// TwinCAT 3 PLC project FlyingSaw
// ProgramVersion: 3.1.4023.0
// libraries:
//   Struckig, * (Stefan Besler)
//   Tc3_Module, * (Beckhoff Automation GmbH)
//   ZApplication, 1.5.37.1 (Zeugwerk GmbH)
//   ZEquipment, 1.5.37.1 (Zeugwerk GmbH)
//   ZAux, 1.5.37.1 (Zeugwerk GmbH)
//   ZPlatform, 1.5.37.1 (Zeugwerk GmbH)
//   ZCore, 1.5.37.1 (Zeugwerk GmbH)
// project tree:
//   ZApp/App/ ZApp.TcPOU
//   ZApp/App/_DataTypes/ ZAppStep.TcDUT
//   ZApp/App/_States/ ZAppSequenceBoot.TcPOU, ZAppSequenceBootFault.TcPOU, ZAppSequenceRunning.TcPOU
//   ZApp/App/_SubObjects/ ZAppSequence.TcPOU
//   ZApp/Com/_DataTypes/ BoxesCom.TcDUT, ZCom.TcDUT, ZComUnit.TcDUT
//   ZApp/Data/_DataTypes/ ZData.TcDUT, ZDataMachine.TcDUT, ZDataConfig.TcDUT, ZDataCalibration.TcDUT, ZDataRecipe.TcDUT
//   ZApp/Unit/Machine/ IMachine.TcIO, MachineUnit.TcPOU, MachineUnitProgram.TcPOU
//   ZApp/Unit/Machine/_Com/ MachineCom.TcDUT, MachineComPublish.TcDUT, MachineComPublishEquipment.TcDUT, MachineComRef.TcDUT, MachineComRequest.TcDUT, MachineComSubscribe.TcDUT, MachineComSubscribeEquipment.TcDUT
//   ZApp/Unit/Machine/_DataTypes/ Box.TcDUT, MachineState.TcDUT, MachineStep.TcDUT
//   ZApp/Unit/Machine/_Data/ MachineDataCalibration.TcDUT, MachineDataConfig.TcDUT, MachineDataMachine.TcDUT, MachineDataRef.TcDUT
//   ZApp/Unit/Machine/_Equipment/ MachineActuator.TcPOU, MachineAxis.TcPOU, MachineEquipment.TcPOU, MachineFieldbus.TcPOU, MachineIo.TcPOU, MachineLinkedUnit.TcPOU
//   ZApp/Unit/Machine/_States/ MachineSequenceAutomatic.TcPOU, MachineSequenceBoot.TcPOU, MachineSequenceFaultReaction.TcPOU, MachineSequenceGoHome.TcPOU, MachineSequenceStop.TcPOU
//   ZApp/Unit/Machine/_SubObjects/ BoxRingBuffer.TcPOU, MachineContainer.TcPOU, MachineSequence.TcPOU
//   ZApp/ ZGlobal.TcGVL, ZModuleProgram.TcPOU, ZModuleTask.TcTTO
// real-time tasks:
//   TASK ZModuleTask: cycle T#10ms, priority 20, ADS port 350

CONFIGURATION FlyingSaw
    RESOURCE PLC ON TwinCAT3
        TASK ZModuleTask(INTERVAL := T#10ms, PRIORITY := 20);
        PROGRAM ZModuleProgram WITH ZModuleTask : ZModuleProgram;
    END_RESOURCE
END_CONFIGURATION

// ---- ZApp/App/_DataTypes/ZAppStep.TcDUT
{attribute 'qualified_only'}
{attribute 'to_string'}
TYPE ZAppStep :
(
  Undefined := 0
  
  ,BootBegin
  ,BootLoadDefaultData
  ,BootEnd
  ,BootFaultBegin
  ,BootFaultEnd 
  ,RunningBegin
  ,RunningEnd   
);
END_TYPE

// ---- ZApp/Com/_DataTypes/BoxesCom.TcDUT
TYPE BoxesCom :
STRUCT
  IndexOfFirst : DINT;
  IndexOfNext : DINT;
  Buffer : ARRAY [0..20] OF Box;
END_STRUCT
END_TYPE

// ---- ZApp/Com/_DataTypes/ZCom.TcDUT
TYPE ZCom :
STRUCT
  // module context
  App : ZApplication.ApplicationComPublish;
  Alarming : ZApplication.AlarmingCom;
  Messages : ZApplication.MessagingCom;
  
  // unit context
  Unit : ZComUnit;
  
  Boxes : BoxesCom;

END_STRUCT
END_TYPE

// ---- ZApp/Com/_DataTypes/ZComUnit.TcDUT
TYPE ZComUnit :
STRUCT
{region "Machine"}
{IF NOT (defined (Machine_disabled))}
  Machine : MachineCom;
  {attribute 'ZId' := 'ffcc16ae-32b8-4aad-8514-f391c00062a3'}
{END_IF}
{endregion}
{attribute '__ZwPlcApplicationComUnitDeclaration__'} // Do not remove this attribute! It is used for code generation.
END_STRUCT
END_TYPE

// ---- ZApp/Data/_DataTypes/ZData.TcDUT
TYPE ZData :
STRUCT
  Config : ZDataConfig;
  Machine : ZDataMachine;
  Calibration : ZDataCalibration;
  Recipe : ZDataRecipe;
END_STRUCT
END_TYPE

// ---- ZApp/Data/_DataTypes/ZDataMachine.TcDUT
TYPE ZDataMachine :
STRUCT
{region "Machine"}
{IF NOT (defined (Machine_disabled))}
  Machine : MachineDataMachine;
  {attribute 'ZId' := 'ffcc16ae-32b8-4aad-8514-f391c00062a3'}
{END_IF}
{endregion}
{attribute '__ZwPlcApplicationDataMachineDeclaration__'} // Do not remove this attribute! It is used for code generation.
END_STRUCT
END_TYPE

// ---- ZApp/Data/_DataTypes/ZDataConfig.TcDUT
TYPE ZDataConfig :
STRUCT
{region "Machine"}
{IF NOT (defined (Machine_disabled))}
  Machine : MachineDataConfig;
  {attribute 'ZId' := 'ffcc16ae-32b8-4aad-8514-f391c00062a3'}
{END_IF}
{endregion}
{attribute '__ZwPlcApplicationDataConfigDeclaration__'} // Do not remove this attribute! It is used for code generation.
END_STRUCT
END_TYPE

// ---- ZApp/Data/_DataTypes/ZDataCalibration.TcDUT
TYPE ZDataCalibration :
STRUCT
{region "Machine"}
{IF NOT (defined (Machine_disabled))}
  Machine : MachineDataCalibration;
  {attribute 'ZId' := 'ffcc16ae-32b8-4aad-8514-f391c00062a3'}
{END_IF}
{endregion}
{attribute '__ZwPlcApplicationDataCalibrationDeclaration__'} // Do not remove this attribute! It is used for code generation.
END_STRUCT
END_TYPE

// ---- ZApp/Data/_DataTypes/ZDataRecipe.TcDUT
TYPE ZDataRecipe :
STRUCT
  RecipeParam1 : LREAL;
  RecipeParam2 : LREAL;
  RecipeParam3 : LREAL;
END_STRUCT
END_TYPE

// ---- ZApp/Unit/Machine/_Com/MachineCom.TcDUT
/// This struct contains variables that
/// * are read from outside (e.g. HMI) to retrieve information about the unit's current state and (temporary) parameters (= `publish`) 
/// * are written from outside (e.g. HMI) to control the unit via ADS (= `subscribe`) 
TYPE MachineCom :
STRUCT
  Publish : MachineComPublish;
  Subscribe : MachineComSubscribe;
END_STRUCT
END_TYPE

// ---- ZApp/Unit/Machine/_Com/MachineComPublish.TcDUT
/// this is the container of informations that the unit wants to share with the world outside of the PLC
/// This struct should only be read from by external applications.
TYPE MachineComPublish :
STRUCT
  State : ZApplication.UnitStateMachineState; // state the unit is in
  Request : MachineComRequest; // booleans that indictate which action is currently possible to perform with this unit
  Equipment : MachineComPublishEquipment;  // structs for equipment objects which are used by the bridges
END_STRUCT
END_TYPE

// ---- ZApp/Unit/Machine/_Com/MachineComPublishEquipment.TcDUT
TYPE MachineComPublishEquipment :
STRUCT

{region "TransportX : Axis"}
  TransportX : ZApplication.AxisComPublish;
  {attribute 'ZId' := 'e985697b-7ba2-4e1b-acce-25e7c1308b60'}
{endregion}

{region "ToolX : Axis"}
  ToolX : ZApplication.AxisComPublish;
  {attribute 'ZId' := '805b377d-816e-493b-a105-09954c5e25a1'}
{endregion}

{attribute '__ZwPlcUnitComDeclaration__'} // Do not remove this attribute! It is used for code generation.

END_STRUCT
END_TYPE

// ---- ZApp/Unit/Machine/_Com/MachineComRef.TcDUT
/// container for all communication data types that are used by the unit
TYPE MachineComRef :
STRUCT
  Publish : REFERENCE TO MachineComPublish; 
  Subscribe : REFERENCE TO MachineComSubscribe; 
END_STRUCT
END_TYPE

// ---- ZApp/Unit/Machine/_Com/MachineComRequest.TcDUT
TYPE MachineComRequest :
STRUCT
  Start : BOOL;
  Stop : BOOL;
  GoHome : BOOL;
  Halt : BOOL;
END_STRUCT
END_TYPE

// ---- ZApp/Unit/Machine/_Com/MachineComSubscribe.TcDUT
TYPE MachineComSubscribe :
STRUCT
  Request : MachineComRequest; // contains booleans that are used to start a specific sequence.
  Equipment : MachineComSubscribeEquipment;  // structs for equipment objects which are used by the bridges
END_STRUCT
END_TYPE

// ---- ZApp/Unit/Machine/_Com/MachineComSubscribeEquipment.TcDUT
TYPE MachineComSubscribeEquipment :
STRUCT

{region "TransportX : Axis"}
  TransportX : ZApplication.AxisComSubscribe;
  {attribute 'ZId' := 'e985697b-7ba2-4e1b-acce-25e7c1308b60'}
{endregion}

{region "ToolX : Axis"}
  ToolX : ZApplication.AxisComSubscribe;
  {attribute 'ZId' := '805b377d-816e-493b-a105-09954c5e25a1'}
{endregion}

{region "BoxDetected : Digital"}
  BoxDetected : ZApplication.DigitalComSubscribe;
  {attribute 'ZId' := 'd9755a0b-6503-481c-99e0-54f892b6c08c'}
{endregion}

{attribute '__ZwPlcUnitComDeclaration__'} // Do not remove this attribute! It is used for code generation.

END_STRUCT
END_TYPE

// ---- ZApp/Unit/Machine/_DataTypes/Box.TcDUT
TYPE Box :
STRUCT
  BoxId : INT;
  DetectedAt : LWORD;
  CompletionRatio : LREAL;
END_STRUCT
END_TYPE

// ---- ZApp/Unit/Machine/_DataTypes/MachineState.TcDUT
/// This enumeration contains all used defined sequences of a unit.
/// Per default a unit makes use of the states that are contained in (UnitStateDefault)[xref:ZApplication.UnitStateDefault]. However,
/// most of the time a unit need to perform some application depend sequences that can be performed by putting the unit into userdefined states.
/// For instance, a robotic unit could use the state (automatic)[xref:ZApplication.UnitStateDefault] to lift an object from point A to point B,
/// a userdefined state could be used to open and close the robotic-units gripper, respectively
{attribute 'qualified_only'}
TYPE MachineState :
(
	UserdefinedState1 := ZApplication.UnitStateMachineState.Last+1
);
END_TYPE

// ---- ZApp/Unit/Machine/_DataTypes/MachineStep.TcDUT
/// This enumeration contains all steps that are used by the various sequences of a unit.
/// Sequences use a subrange (***Begin to ***End) of this enumeration.
{attribute 'qualified_only'}
{attribute 'to_string'}
TYPE MachineStep :
(
  Undefined := 0
  
  ,BootBegin
  ,BootEnd 

  ,StopBegin
  ,StopEnd

  ,AutomaticBegin
  ,AutomaticRunTool
  ,AutomaticEnd
  
  ,GoHomeBegin
  ,GoHomeEnd 
  
  ,FaultReactionBegin
  ,FaultReactionEnd
);
END_TYPE

// ---- ZApp/Unit/Machine/_Data/MachineDataCalibration.TcDUT
/// calibration that is determined by calibration sequences of the unit (static offsets, shifts)
TYPE MachineDataCalibration :
STRUCT
END_STRUCT
END_TYPE

// ---- ZApp/Unit/Machine/_Data/MachineDataConfig.TcDUT
/// configuration data that is used during boot to configure the Units equipment
TYPE MachineDataConfig :
STRUCT
  Simulated : BOOL;
END_STRUCT
END_TYPE

// ---- ZApp/Unit/Machine/_Data/MachineDataMachine.TcDUT
/// machine data that is used through most sequences of the unit (motor speed, axes positions, ...)
TYPE MachineDataMachine :
STRUCT
  Slowspeed : LREAL;
  Highspeed : LREAL;
END_STRUCT
END_TYPE

// ---- ZApp/Unit/Machine/_Data/MachineDataRef.TcDUT
/// container for all data that are used by the unit
TYPE MachineDataRef :
STRUCT
  Config : REFERENCE TO MachineDataConfig; // data required for booting the unit (axes configuration, simulation, parameters that have to be written in PREOP, ...)
  Machine : REFERENCE TO MachineDataMachine; // speeds, positions, ...
  Calibration : REFERENCE TO MachineDataCalibration; // offsets, shifts of nominal to actual values
END_STRUCT
END_TYPE

// ---- ZApp/ZGlobal.TcGVL
{attribute 'qualified_only'}
VAR_GLOBAL
  Com : ZCom;
END_VAR
VAR_GLOBAL PERSISTENT
  Data : ZData;
END_VAR

// ---- ZApp/Unit/Machine/IMachine.TcIO
INTERFACE IMachine EXTENDS ZApplication.IUnit

END_INTERFACE

// ---- ZApp/ZModuleProgram.TcPOU
/// Zeugwerk Application
PROGRAM ZModuleProgram
VAR_INPUT
{region "ZModuleProgram : Utility"}
  App : ZApp(displayName:='Zeugwerk-Application Template', com:=ZGlobal.Com.App);
  Datetime : ZAux.DateTimeUM;
  {attribute 'ZId' := ''}
{endregion}
{region "ZModuleProgram : Logging"}
  Alarming : ZApplication.Alarming(App, datetime := Datetime, com := ZGlobal.Com.Alarming);
  LoggerHmi : ZApplication.Messaging(App, datetime := Datetime, com := ZGlobal.Com.Messages);
  LoggerFile : ZAux.LoggerFile7FF(App, datetime := Datetime, filePath:='C:\Zeugwerk\logs\messages.log', target:='');
  Logger : ZAux.Logging;
  {attribute 'ZId' := ''}
{endregion}  
{attribute '__ZwPlcApplicationModuleProgramDeclaration__'} // Do not remove this attribute! It is used for code generation.
{region "Machine"}
{undefine RunInSeparateProgram}
{IF NOT (defined (Machine_disabled)) AND NOT (defined (RunInSeparateProgram))}
  Machine : MachineUnit(name := 'Machine', // name of the unit (for logging)
					  parent := App, // caller of the Unit's cyclic method. If the Unit runs in its own context use 0
						configdata := ZGlobal.Data.Config.Machine,
						machinedata := ZGlobal.Data.Machine.Machine,
						calibrationdata := ZGlobal.Data.Calibration.Machine,
						com := ZGlobal.Com.Unit.Machine);
  {attribute 'section' := '__ZwPlcUnitProgramDeclaration__'}
  {attribute 'ZId' := 'ffcc16ae-32b8-4aad-8514-f391c00062a3'}
{END_IF}
{endregion}
{attribute '__ZwPlcUnitProgramDeclaration__'} // Do not remove this attribute! It is used for code generation.
END_VAR

{region "ZModuleProgram : Utility"}
  Datetime.Cyclic();
  App.Cyclic();
  {attribute 'ZId' := ''}
{endregion}
{attribute '__ZwPlcApplicationModuleProgramImplementation__'} // Do not remove this attribute! It is used for code generation.

END_PROGRAM

// ---- ZApp/App/ZApp.TcPOU
FUNCTION_BLOCK ZApp EXTENDS ZApplication.Application
VAR
  _boot : ZAppSequenceBoot;
  _bootFault : ZAppSequenceBootFault;
  _running : ZAppSequenceRunning;
END_VAR

METHOD FB_init : BOOL
VAR_INPUT
  bInitRetains : BOOL; /// if TRUE, the retain variables are initialized (warm start / cold start)
  bInCopyCode : BOOL; /// if TRUE, the instance afterwards gets moved into the copy code (online change)
  displayName : ZCore.ZString;
  com : REFERENCE TO ZApplication.ApplicationComPublish;
END_VAR
SetBootSequence(_boot);
SetBootFaultSequence(_bootFault);
SetRunningSequence(_running);
END_METHOD

END_FUNCTION_BLOCK

// ---- ZApp/App/_States/ZAppSequenceBoot.TcPOU
FUNCTION_BLOCK ZAppSequenceBoot EXTENDS ZAppSequence IMPLEMENTS ZCore.ISequence
VAR
  _step : ZCore.Step(ZAppStep.BootBegin, ZAppStep.BootEnd);
END_VAR

IF OnStart(_step)
THEN
  // init custom sequence variables here ...
END_IF

REPEAT
  LogStep();

  CASE _step.Index OF
    (* -------------------------------------------------------------------------------------------------------------------------------- *)
    ZAppStep.BootBegin:
    (* -------------------------------------------------------------------------------------------------------------------------------- *)
    
      IF _step.OnEntry()
      THEN
        ZModuleProgram.LoggerFile.MinimumLevel := ZCore.LogLevel.Trace;
        ZModuleProgram.Logger.AddLogger(ZModuleProgram.LoggerFile);        
        {attribute '__ZwPlcAppZComModuleContext__'} // Do not remove this attribute! It is used for code generation.      
      END_IF
      
	  IF ZModuleProgram.Datetime.State <> ZCore.ObjectState.Booting
      THEN
        _step.SetNext(ZAppStep.BootLoadDefaultData);        
      END_IF
      
    (* -------------------------------------------------------------------------------------------------------------------------------- *)
    ZAppStep.BootLoadDefaultData:
    (* -------------------------------------------------------------------------------------------------------------------------------- *)

      {warning 'The application is loading the default config data on every restart!'}
      LoadDefaultConfigData();
      
      IF IsCommissioning()
      THEN
        LoadDefaultData();
      END_IF
      
      _step.SetNext(ZAppStep.BootEnd);
      
    (* -------------------------------------------------------------------------------------------------------------------------------- *)
    ZAppStep.BootEnd:
    (* -------------------------------------------------------------------------------------------------------------------------------- *)
      SetBusy(FALSE);
      
  ELSE
    Abort('sequence contains unhandled step');
  END_CASE
UNTIL _step.IsNotRepeatable() OR_ELSE NOT Busy END_REPEAT

METHOD  IsCommissioning : BOOL
IsCommissioning := TRUE;
END_METHOD

METHOD FINAL LoadDefaultConfigData

{region "Machine"}
  {IF NOT (defined (Machine_disabled))}
  ZGlobal.Data.Config.Machine.Simulated := TRUE;
  {region "UserInitCode"}
  // put your individual init code for this unit here
  {endregion}
  {END_IF}
  {attribute 'ZId' := 'ffcc16ae-32b8-4aad-8514-f391c00062a3'}
{endregion}

{attribute '__ZwPlcUnitLoadDefaultConfigData__'} // Do not remove this attribute! It is used for code generation.
END_METHOD

METHOD FINAL LoadDefaultData

{attribute '__ZwPlcUnitLoadDefaultData__'} // Do not remove this attribute! It is used for code generation.
END_METHOD

END_FUNCTION_BLOCK

// ---- ZApp/App/_SubObjects/ZAppSequence.TcPOU
FUNCTION_BLOCK ABSTRACT ZAppSequence EXTENDS ZApplication.Sequence IMPLEMENTS ZCore.ISequence

METHOD StepDecoded : ZCore.ZString
VAR_INPUT
  stepIndex : INT;
END_VAR
VAR_INST
  _stepIndexDecoded : ZAppStep;
END_VAR
_stepIndexDecoded := stepIndex;
StepDecoded := TO_STRING(_stepIndexDecoded);
END_METHOD

END_FUNCTION_BLOCK

// ---- ZApp/App/_States/ZAppSequenceBootFault.TcPOU
FUNCTION_BLOCK ZAppSequenceBootFault EXTENDS ZAppSequence IMPLEMENTS ZCore.ISequence
VAR
  _step : ZCore.Step(ZAppStep.BootFaultBegin, ZAppStep.BootFaultEnd);
END_VAR

IF OnStart(_step)
THEN
  // init custom sequence variables here ...
END_IF

REPEAT
  LogStep();

  CASE _step.Index OF
    (* -------------------------------------------------------------------------------------------------------------------------------- *)
    ZAppStep.BootFaultBegin:
    (* -------------------------------------------------------------------------------------------------------------------------------- *)
      _step.SetNext(ZAppStep.BootFaultEnd);
      
    (* -------------------------------------------------------------------------------------------------------------------------------- *)
    ZAppStep.BootFaultEnd:
    (* -------------------------------------------------------------------------------------------------------------------------------- *)
      SetBusy(FALSE);
      
  ELSE
    Abort('sequence contains unhandled step');
  END_CASE
UNTIL _step.IsNotRepeatable() OR_ELSE NOT Busy END_REPEAT

END_FUNCTION_BLOCK

// ---- ZApp/App/_States/ZAppSequenceRunning.TcPOU
FUNCTION_BLOCK ZAppSequenceRunning EXTENDS ZAppSequence IMPLEMENTS ZCore.ISequence
VAR
  _step : ZCore.Step(ZAppStep.RunningBegin, ZAppStep.RunningEnd);
END_VAR

IF OnStart(_step)
THEN
  // init custom sequence variables here ...
END_IF

REPEAT
  LogStep();

  CASE _step.Index OF
    (* -------------------------------------------------------------------------------------------------------------------------------- *)
    ZAppStep.RunningBegin:
    (* -------------------------------------------------------------------------------------------------------------------------------- *)
      ; // implement me
      
    (* -------------------------------------------------------------------------------------------------------------------------------- *)
    ZAppStep.RunningEnd:
    (* -------------------------------------------------------------------------------------------------------------------------------- *)
      SetBusy(FALSE);
      
  ELSE
    Abort('sequence contains unhandled step');
  END_CASE
UNTIL _step.IsNotRepeatable() OR_ELSE NOT Busy END_REPEAT

END_FUNCTION_BLOCK

// ---- ZApp/Unit/Machine/MachineUnit.TcPOU
/// Declaration of a distinct unit of this application
FUNCTION_BLOCK MachineUnit EXTENDS ZApplication.Unit IMPLEMENTS IMachine
VAR
  _equipment : MachineEquipment(THIS^);
  _data : MachineDataRef;
  _com : MachineComRef;

  _boot : MachineSequenceBoot(THIS^);
  _automatic : MachineSequenceAutomatic(THIS^);
  _stop : MachineSequenceStop(THIS^);
  _gohome : MachineSequenceGoHome(THIS^);
  _faultReaction : MachineSequenceFaultReaction(THIS^);
  
  _statemachine : ZApplication.UnitStateMachine;

  _observeTimer : ZAux.Timer; 
END_VAR

{attribute 'ZId' := '7a669cb2-1530-4a61-a6bf-785d936ff64f'}

IF _observeTimer.Done THEN
  _observeTimer.WaitAsync(0.1);
  
  // monitor _com for requested actions (e.g. start homing, start automatic mode, ...)
  ObserveRequest(_com.Subscribe.Request.Start, ZApplication.UnitStateMachineState.Automatic);
  ObserveRequest(_com.Subscribe.Request.Stop, ZApplication.UnitStateMachineState.Stop);
  ObserveRequest(_com.Subscribe.Request.GoHome, ZApplication.UnitStateMachineState.GoHome);
  ObserveRequest(_com.Subscribe.Request.Halt, ZApplication.UnitStateMachineState.Halt);
  
  // provide relevant information via ADS
  _com.Publish.Request.Stop := _stateMachine.IsTransitionAllowed(ZApplication.UnitStateMachineState.Stop);
  _com.Publish.Request.Start := _stateMachine.IsTransitionAllowed(ZApplication.UnitStateMachineState.Automatic);
  _com.Publish.Request.GoHome := _stateMachine.IsTransitionAllowed(ZApplication.UnitStateMachineState.GoHome);
  _com.Publish.Request.Halt := _stateMachine.IsTransitionAllowed(ZApplication.UnitStateMachineState.Halt);

  _com.Publish.State := _stateMachine.State();
END_IF

METHOD FB_init : BOOL
VAR_INPUT
  bInitRetains : BOOL; // if TRUE, the retain variables are initialized (warm start / cold start)
  bInCopyCode : BOOL;  // if TRUE, the instance afterwards gets moved into the copy code (online change)
  parent : ZCore.IManagedObject; // caller of the Unit's cyclic method. If the Unit runs in its own context use 0
  name : ZCore.ZString;  // name of this unit as it should show up in the logger
  configdata : REFERENCE TO MachineDataConfig;  // reference to the configuration data that is used during boot to configure the Units equipment
  machinedata : REFERENCE TO MachineDataMachine; // reference to the machine data that is used through most sequences of the unit (motor speed, axes positions, ...)
  calibrationdata : REFERENCE TO MachineDataCalibration;  // reference to calibration that is determined by calibration sequences of the unit (static offsets, shifts)
  com : REFERENCE TO MachineCom;  // reference to the communication interface that is used to control this Unit via ADS
END_VAR
_name := name;

// initialize local logger decorator
_loggerDecorator.FB_init(bInitRetains, bInCopyCode, name, ZModuleProgram.Logger);
_alarmingDecorator.FB_init(bInitRetains, bInCopyCode, name, ZModuleProgram.Alarming);

// setup data
_data.Config REF= configdata;
_data.Machine REF= machinedata;
_data.Calibration REF= calibrationdata;
_com.Publish REF= com.Publish;
_com.Subscribe REF= com.Subscribe;

// ------- sequence initialization, map sequences of this unit to the statemachine -------
{attribute '__ZwPlcUnitInitSequenceImplementation__'} // Do not remove this attribute! It is used for code generation.
_statemachine.SetSequence(ZApplication.UnitStateMachineState.Boot, _boot);
_statemachine.SetSequence(ZApplication.UnitStateMachineState.FaultReaction, _faultReaction);
_statemachine.SetSequence(ZApplication.UnitStateMachineState.Gohome, _gohome);
_statemachine.SetSequence(ZApplication.UnitStateMachineState.Stop, _stop);
_statemachine.SetSequence(ZApplication.UnitStateMachineState.Automatic, _automatic);

_statemachine.SetName(_name);
_statemachine.SetLogger(_logger);

// set initial state
_statemachine.SetState(ZApplication.UnitStateMachineState.Boot);
SetStateMachine(_statemachine);
END_METHOD

END_FUNCTION_BLOCK

// ---- ZApp/Unit/Machine/_Equipment/MachineEquipment.TcPOU
/// This function block is a container for equipment that is used by this unit.
/// Equipment is grouped by its kind (actuator, axes, io, ...).
/// It extends from [ManagedObjectContainer](xref:ZCore.ManagedObjectContainer) such that the parent
/// (= the unit itself) can be passed to equipment instances.
FUNCTION_BLOCK MachineEquipment EXTENDS MachineContainer
VAR_INPUT
  Io : MachineIo(_parent);
  Actuator : MachineActuator(_parent);
  Axis : MachineAxis(_parent);
  Fieldbus : MachineFieldbus(_parent);
  Unit : MachineLinkedUnit(_parent);
END_VAR

END_FUNCTION_BLOCK

// ---- ZApp/Unit/Machine/_SubObjects/MachineContainer.TcPOU
FUNCTION_BLOCK MachineContainer EXTENDS ZCore.ObjectContainer
VAR_INPUT
END_VAR
VAR_OUTPUT
END_VAR
VAR
  {attribute 'hide'}
  _parent : REFERENCE TO MachineUnit;
END_VAR

{attribute 'hide' }
METHOD FB_init : BOOL
VAR_INPUT
	bInitRetains : BOOL; // if TRUE, the retain variables are initialized (warm start / cold start)
	bInCopyCode : BOOL;  // if TRUE, the instance afterwards gets moved into the copy code (online change)
  unit : REFERENCE TO MachineUnit;
END_VAR
_parent REF= unit;
END_METHOD

END_FUNCTION_BLOCK

// ---- ZApp/Unit/Machine/_Equipment/MachineIo.TcPOU
/// This function block is a container for all I/Os that are used by this unit.
/// The parent of all objects can be directly transfered in their constructor (this is only relevant for equipment objects
/// that have to be managed (e.g. [DebouncedInput](xref:ZEquipment.DebouncedInput), [Light](xref:ZEquipment.Light), ...).
FUNCTION_BLOCK MachineIo EXTENDS MachineContainer
VAR
  {attribute 'hide'}
  _iobridge : ZApplication.IoBridge(_parent);
END_VAR
VAR_INPUT

{region "BoxDetected : DigitalInput"}
  BoxDetected : ZEquipment.DigitalInput;
  {attribute 'ZId' := 'd9755a0b-6503-481c-99e0-54f892b6c08c'}
{endregion}

{attribute '__ZwPlcUnitEquipmentDeclaration__'} // Do not remove this attribute! It is used for code generation.
END_VAR

IF _isInitialized
THEN
  RETURN;
END_IF

  _iobridge.SetLogger(_parent._logger);

{region "BoxDetected : DigitalInput"}
  BoxDetected.SetLogger(_parent._logger);
  BoxDetected.SetName('BoxDetected');
  BoxDetected.SetSimulation(on:=_parent._data.Config.Simulated);
  BoxDetected.SetLogic(ZEquipment.DigitalLogic.Normal);
  _ioBridge.AddDigitalInput(BoxDetected, publish := _parent._com.Publish.Equipment.BoxDetected, subscribe := _parent._com.Subscribe.Equipment.BoxDetected);

  {region "UserInitCode"}
  // put your individual init code for this I/O here
  {endregion}

  {attribute 'ZId' := 'd9755a0b-6503-481c-99e0-54f892b6c08c'}
{endregion}

{attribute '__ZwPlcUnitEquipmentImplementation__'} // Do not remove this attribute! It is used for code generation.

_isInitialized := TRUE;

END_FUNCTION_BLOCK

// ---- ZApp/Unit/Machine/_Equipment/MachineActuator.TcPOU
/// This function block is a container for all actuator objects that are used by this unit.
/// The parent of all objects can be directly transfered in their constructor (this is only relevant for equipment objects
/// that have to be managed (e.g. [DebouncedInput](xref:ZEquipment.DebouncedInput), [Light](xref:ZEquipment.Light), ...).
FUNCTION_BLOCK MachineActuator EXTENDS MachineContainer
VAR
  {attribute 'hide'}
  _actuatorbridge : ZApplication.ActuatorBridge(_parent);
  {attribute 'hide'}
  _iobridge : ZApplication.IoBridge(_parent);
END_VAR
VAR_INPUT

{attribute '__ZwPlcUnitEquipmentDeclaration__'} // Do not remove this attribute! It is used for code generation.
END_VAR

IF _isInitialized
THEN
  RETURN;
END_IF

  _actuatorbridge.SetLogger(_parent._logger);

{attribute '__ZwPlcUnitEquipmentImplementation__'} // Do not remove this attribute! It is used for code generation.

_isInitialized := TRUE;

END_FUNCTION_BLOCK

// ---- ZApp/Unit/Machine/_Equipment/MachineAxis.TcPOU
/// This function block is a container for all axis objects that are used by this unit.
/// The parent of all objects can be directly transfered in their constructor (this is only relevant for equipment objects
/// that have to be managed (e.g. [DebouncedInput](xref:ZEquipment.DebouncedInput), [Light](xref:ZEquipment.Light), ...).
FUNCTION_BLOCK MachineAxis EXTENDS MachineContainer
VAR
  {attribute 'hide'}
  _axisbridge : ZApplication.AxisBridge(_parent);
END_VAR
VAR_INPUT

{region "TransportX : AxisPlcOpenMc"}
  TransportX : ZEquipment.AxisSimulated(_parent);
  {attribute 'ZId' := 'e985697b-7ba2-4e1b-acce-25e7c1308b60'}
{endregion}

{region "ToolX : AxisPlcOpenMc"}
  ToolX : ZEquipment.AxisSimulated(_parent);
  {attribute 'ZId' := '805b377d-816e-493b-a105-09954c5e25a1'}
{endregion}

{attribute '__ZwPlcUnitEquipmentDeclaration__'} // Do not remove this attribute! It is used for code generation.
END_VAR

IF _isInitialized
THEN
  RETURN;
END_IF

  _axisbridge.SetLogger(_parent._logger);

{region "TransportX : AxisPlcOpenMc"}
  TransportX.SetLogger(_parent._logger);
  TransportX.SetName(name:='TransportX');
  TransportX.SetSimulation(_parent._data.Config.Simulated);
  _axisbridge.WithHoming(TransportX)
     .WithMovePosition(TransportX)
     .WithMoveVelocity(TransportX)
     .WithHalt(TransportX)
     .WithVelocityFeedrate(TransportX)
     .WithFeedbackPosition(TransportX)
     .WithFeedbackVelocity(TransportX)
     .WithFeedbackCurrent(TransportX)
     .AddAxis (axis:=TransportX, publish:=_parent._com.Publish.Equipment.TransportX, subscribe:=_parent._com.Subscribe.Equipment.TransportX);


  {region "UserInitCode"}
  // put your individual init code for this Axis here
  {endregion}

  {attribute 'ZId' := 'e985697b-7ba2-4e1b-acce-25e7c1308b60'}
{endregion}

{region "ToolX : AxisPlcOpenMc"}
  ToolX.SetLogger(_parent._logger);
  ToolX.SetName(name:='ToolX');
  ToolX.SetSimulation(_parent._data.Config.Simulated);
  _axisbridge.WithHoming(ToolX)
     .WithMovePosition(ToolX)
     .WithMoveVelocity(ToolX)
     .WithHalt(ToolX)
     .WithVelocityFeedrate(ToolX)
     .WithFeedbackPosition(ToolX)
     .WithFeedbackVelocity(ToolX)
     .WithFeedbackCurrent(ToolX)
     .AddAxis (axis:=ToolX, publish:=_parent._com.Publish.Equipment.ToolX, subscribe:=_parent._com.Subscribe.Equipment.ToolX);

  {region "UserInitCode"}
  // put your individual init code for this Axis here
  {endregion}

  {attribute 'ZId' := '805b377d-816e-493b-a105-09954c5e25a1'}
{endregion}

{attribute '__ZwPlcUnitEquipmentImplementation__'} // Do not remove this attribute! It is used for code generation.

_isInitialized := TRUE;

END_FUNCTION_BLOCK

// ---- ZApp/Unit/Machine/_Equipment/MachineFieldbus.TcPOU
/// This function block is a container for all axis objects that are used by this unit.
/// The parent of all objects can be directly transfered in their constructor (this is only relevant for equipment objects
/// that have to be managed (e.g. [DebouncedInput](xref:ZEquipment.DebouncedInput), [Light](xref:ZEquipment.Light), ...).
FUNCTION_BLOCK MachineFieldbus EXTENDS MachineContainer
VAR
END_VAR
VAR_INPUT

{attribute '__ZwPlcUnitEquipmentDeclaration__'} // Do not remove this attribute! It is used for code generation.
END_VAR

IF _isInitialized
THEN
  RETURN;
END_IF

{attribute '__ZwPlcUnitEquipmentImplementation__'} // Do not remove this attribute! It is used for code generation.

_isInitialized := TRUE;

END_FUNCTION_BLOCK

// ---- ZApp/Unit/Machine/_Equipment/MachineLinkedUnit.TcPOU
/// This function block is a container for all linked units that are used by this unit.
/// Linked units can be addressed through their individual interface.
FUNCTION_BLOCK MachineLinkedUnit EXTENDS MachineContainer
VAR_INPUT
{attribute '__ZwPlcUnitEquipmentDeclaration__'} // Do not remove this attribute! It is used for code generation.
END_VAR

IF _isInitialized
THEN
  RETURN;
END_IF

{attribute '__ZwPlcUnitEquipmentImplementation__'} // Do not remove this attribute! It is used for code generation.

_isInitialized := TRUE;

END_FUNCTION_BLOCK

// ---- ZApp/Unit/Machine/_States/MachineSequenceBoot.TcPOU
FUNCTION_BLOCK MachineSequenceBoot EXTENDS MachineSequence IMPLEMENTS ZCore.ISequence
VAR
  _step : ZCore.Step(MachineStep.BootBegin, MachineStep.BootEnd);
END_VAR

IF OnStart(_step) THEN
  ; // init custom sequence variables here ...
END_IF

REPEAT
  LogStep();

  CASE _step.Index OF
    (* -------------------------------------------------------------------------------------------------------------------------------- *)
    MachineStep.BootBegin:
    (* -------------------------------------------------------------------------------------------------------------------------------- *)
      IF _step.OnEntry()
      THEN
        // initialize equipment
        _io();
        _actuator();
        _fieldbus();
        _axis();
        _unit();
      END_IF
      
      _parent._objectManager.Cyclic();      
      Assert(_parent._objectManager);
      IF _parent._objectManager.Booted
      THEN
        _step.SetNext(MachineStep.BootEnd);
      END_IF

    (* -------------------------------------------------------------------------------------------------------------------------------- *)
    MachineStep.BootEnd:
    (* -------------------------------------------------------------------------------------------------------------------------------- *)
      SetBusy(FALSE);
      
  ELSE
    Abort('sequence contains unhandled step');
  END_CASE
UNTIL _step.IsNotRepeatable() OR_ELSE NOT Busy END_REPEAT

END_FUNCTION_BLOCK

// ---- ZApp/Unit/Machine/_SubObjects/MachineSequence.TcPOU
FUNCTION_BLOCK MachineSequence EXTENDS ZApplication.Sequence
VAR
  {attribute 'hide'}
  _parent : REFERENCE TO MachineUnit;
  _io : REFERENCE TO MachineIo;
  _actuator : REFERENCE TO MachineActuator;
  _fieldbus : REFERENCE TO MachineFieldbus;
  _axis : REFERENCE TO MachineAxis;
  _data : REFERENCE TO MachineDataRef;
  _unit : REFERENCE TO MachineLinkedUnit;  
END_VAR

METHOD FB_init : BOOL
VAR_INPUT
  bInitRetains : BOOL; // if TRUE, the retain variables are initialized (warm start / cold start)
  bInCopyCode : BOOL;  // if TRUE, the instance afterwards gets moved into the copy code (online change)
  unit : REFERENCE TO MachineUnit;
END_VAR
_parent REF= unit;
_alarming := unit._alarming;
_io REF= unit._equipment.Io;
_actuator REF= unit._equipment.Actuator;
_fieldbus REF= unit._equipment.Fieldbus;
_axis REF= unit._equipment.Axis;
_unit REF= unit._equipment.Unit;
_data REF= unit._data;
_loggerDiagnostics.SetLogger(unit._logger);
END_METHOD

METHOD StepDecoded : ZCore.ZString
VAR_INPUT
  stepIndex : INT;
END_VAR
VAR_INST
  _stepIndexDecoded : MachineStep;
END_VAR
_stepIndexDecoded := stepIndex;
stepDecoded := TO_STRING(_stepIndexDecoded);
END_METHOD

END_FUNCTION_BLOCK

// ---- ZApp/Unit/Machine/_States/MachineSequenceAutomatic.TcPOU
FUNCTION_BLOCK MachineSequenceAutomatic EXTENDS MachineSequence IMPLEMENTS ZCore.ISequence
VAR
  _step : ZCore.Step(MachineStep.AutomaticBegin, MachineStep.AutomaticEnd);
  _timer : ZAux.Timer;
  
  _boxDetectionTimer : ZAux.Timer;
  _boxes : BoxRingBuffer(20, ADR(ZGlobal.Com.Boxes.Buffer));
  _box : REFERENCE TO Box;
  
  _elapsedTime : LREAL;
  _rt : ZAux.RealTime;
  _otg : Struckig.Otg(0, 1);
  _rand : ZAux.RandomUniform(seed:=0, low:=0.1, high:=0.2);
  _moveToBoxDuration : LREAL := 0.5;
  _startToken : ZCore.StartToken;
END_VAR

IF NOT Busy THEN
  RETURN;
END_IF

IF OnStart(_step) THEN
  ; // init custom sequence variables here ...
END_IF

IF OnStop() THEN
  RETURN; // external stop was triggered
END_IF

IF OnHalt() THEN
  ; // Halting := TRUE; // Uncomment to acknowledge that the sequence is halting
END_IF

REPEAT
  LogStep();

  CASE _step.Index OF
    (* -------------------------------------------------------------------------------------------------------------------------------- *)
    MachineStep.AutomaticBegin:
    (* -------------------------------------------------------------------------------------------------------------------------------- *)
      IF _step.OnEntry()
      THEN
        _boxes.SetLogicPtrs(ADR(ZGlobal.Com.Boxes.IndexOfFirst), ADR(ZGlobal.Com.Boxes.IndexOfNext));
        _boxes.Clear();
        
        _axis.TransportX.MoveVelocityAsync(THIS^, _data.Machine.Highspeed);
        _axis.ToolX.MoveInterpolatedPositionAsync(THIS^);
        
        _otg.CycleTime := _rt.CycleTimeInSeconds();
        _otg.ControlInterface := Struckig.ControlInterfaceType.Position;
        _otg.CurrentPosition[0] := _axis.ToolX.ActualPosition;
        _otg.CurrentVelocity[0] := 0;
        _otg.CurrentAcceleration[0] := 0;
     
        _otg.TargetPosition[0] := _otg.CurrentPosition[0];
        _otg.TargetVelocity[0] := 0;
        
        _otg.MaxAcceleration[0] := 30000;
        _otg.MaxJerk[0] := 3000000;
        _otg.MaxVelocity[0] := 1000;
        _otg.EnableAutoPropagate := TRUE;
			END_IF

      Await2(obj1:=_axis.TransportX, obj2:=_axis.ToolX, nextStep:=MachineStep.AutomaticWaitBox);

    (* -------------------------------------------------------------------------------------------------------------------------------- *)
    MachineStep.AutomaticWaitBox:
    (* -------------------------------------------------------------------------------------------------------------------------------- *)
      
      IF _boxes.Size > 0
      THEN
        _box REF= _boxes.Front();
        _step.SetNext(MachineStep.AutomaticMoveToBox);        
			ELSE
        _otg.ControlInterface := Struckig.ControlInterfaceType.Position;
        _otg.TargetPosition[0] := 0;
        _otg.TargetVelocity[0] := 0;
      END_IF
      
    (* -------------------------------------------------------------------------------------------------------------------------------- *)
    MachineStep.AutomaticMoveToBox:
    (* -------------------------------------------------------------------------------------------------------------------------------- *)
      IF _step.OnEntry()
      THEN
        _otg.ControlInterface := Struckig.ControlInterfaceType.Position;
        _elapsedTime := LWORD_TO_LREAL(Now() - _box.DetectedAt) / 1000;
        _otg.TargetPosition[0] := _data.Machine.Highspeed * _moveToBoxDuration + _data.Machine.Highspeed * _elapsedTime;
        _otg.TargetVelocity[0] := _data.Machine.Highspeed;
        _otg.MinDuration := _moveToBoxDuration;
        
      ELSIF _otg.State = Struckig.TrajectoryState.Error
      THEN
        Abort(_otg.ErrorMessage());
      ELSIF _otg.State = Struckig.TrajectoryState.Idle
      THEN
        _step.SetNext(MachineStep.AutomaticMoveWithBox);
      END_IF

    (* -------------------------------------------------------------------------------------------------------------------------------- *)
    MachineStep.AutomaticMoveWithBox:
    (* -------------------------------------------------------------------------------------------------------------------------------- *)
      IF _step.OnEntry()
      THEN        
        _timer.WaitAsync(1.5);
      END_IF
      
      _box.CompletionRatio := _timer.ElapsedTimeNormalized();
      
      Await(obj1:=_timer, nextStep:=MachineStep.AutomaticWaitBox);
      
      IF _timer.Done
      THEN
        _boxes.PopFirstItem();
			END_IF

    (* -------------------------------------------------------------------------------------------------------------------------------- *)
    MachineStep.AutomaticEnd:
    (* -------------------------------------------------------------------------------------------------------------------------------- *)
      SetBusy(FALSE);
  
  ELSE
    Abort('sequence contains unhandled step');
  END_CASE
UNTIL _step.IsNotRepeatable() OR_ELSE NOT Busy END_REPEAT

// Update trajactory
IF _step.Index >= MachineStep.AutomaticWaitBox
THEN
  _otg();
  
  IF _otg.State = Struckig.TrajectoryState.Error
  THEN
    Abort(_otg.ErrorMessage());
  END_IF
  
  _axis.ToolX.SetInterpolatedPosition(startToken:=_startToken, _otg.CurrentPosition[0]);
  _axis.ToolX.SetInterpolatedVelocity(startToken:=_startToken, _otg.CurrentVelocity[0]);
END_IF

// check for incoming boxes
IF _io.BoxDetected.RisingTrigger()
THEN
  _boxes.Append();  
END_IF

METHOD Now : LWORD
VAR_INPUT
END_VAR
Now := ZModuleProgram.Datetime.UnixTimestamp();
END_METHOD

END_FUNCTION_BLOCK

// ---- ZApp/Unit/Machine/_SubObjects/BoxRingBuffer.TcPOU
FUNCTION_BLOCK BoxRingBuffer EXTENDS RingBuffer
VAR
  _bufferPtr : POINTER TO Box;  
END_VAR
VAR_STAT
  BoxId : INT := 1;
END_VAR

METHOD Append
VAR
  i : DINT;
END_VAR
i := IndexOfNextItem();

_bufferPtr[i].BoxId := THIS^.BoxId;
_bufferPtr[i].DetectedAt := ZModuleProgram.Datetime.UnixTimestamp();
_bufferPtr[i].CompletionRatio := 0;

AppendIndex();

THIS^.BoxId := THIS^.BoxId + 1;
IF THIS^.BoxId > 999
THEN
  THIS^.BoxId := 1;
END_IF
END_METHOD

/// Initializes the RingBuffer at construction time of the object by providing the bufferSize.
/// It also inidializes the pointers of head and tail with an internally stored variable.
METHOD FB_init : BOOL
VAR_INPUT
  bInitRetains : BOOL; //< if TRUE, the retain variables are initialized (warm start / cold start)
  bInCopyCode : BOOL; //< if TRUE, the instance afterwards gets moved into the copy code (online change)
  bufferSize : DINT; //< size of the **managable** buffer. The actual databuffer needs to be one element larger than bufferSize, i.e. data : ARRAY[0..bufferSize] OF ???
  bufferPtr : POINTER TO Box;
END_VAR
_bufferPtr := bufferPtr;
END_METHOD

METHOD Front : REFERENCE TO Box
VAR_INPUT
END_VAR
IF NOT THIS^.Empty
THEN
  Front REF= _bufferPtr[THIS^.IndexOfFirstItem()];
END_IF
END_METHOD

END_FUNCTION_BLOCK

// ---- ZApp/Unit/Machine/_States/MachineSequenceStop.TcPOU
FUNCTION_BLOCK MachineSequenceStop EXTENDS MachineSequence IMPLEMENTS ZCore.ISequence
VAR
  _step : ZCore.Step(MachineStep.StopBegin, MachineStep.StopEnd);
  _timerSim : ZAux.Timer;
END_VAR

IF OnStart(_step) THEN
  ; // init custom sequence variables here ...
END_IF

REPEAT
  LogStep();

  CASE _step.Index OF
    (* -------------------------------------------------------------------------------------------------------------------------------- *)
    MachineStep.StopBegin:
    (* -------------------------------------------------------------------------------------------------------------------------------- *)
      IF _step.OnEntry()
      THEN
        _axis.ToolX.StopAsync(THIS^);
        _axis.TransportX.StopAsync(THIS^);  
			END_IF
      
      Await2(obj1:=_axis.ToolX, obj2:=_axis.TransportX, nextStep:=MachineStep.StopEnd);

    (* -------------------------------------------------------------------------------------------------------------------------------- *)
    MachineStep.StopEnd:
    (* -------------------------------------------------------------------------------------------------------------------------------- *)    
      SetBusy(FALSE);
  
  ELSE
    Abort('sequence contains unhandled step');
  END_CASE
UNTIL _step.IsNotRepeatable() OR_ELSE NOT Busy END_REPEAT

END_FUNCTION_BLOCK

// ---- ZApp/Unit/Machine/_States/MachineSequenceGoHome.TcPOU
FUNCTION_BLOCK MachineSequenceGoHome EXTENDS MachineSequence IMPLEMENTS ZCore.ISequence
VAR
  _step : ZCore.Step(MachineStep.GohomeBegin, MachineStep.GohomeEnd);
  _timer : ZAux.Timer;
END_VAR

IF NOT Busy THEN
  RETURN;
END_IF

IF OnStart(_step) THEN
  ; // init custom sequence variables here ...
END_IF

IF OnStop() THEN
  RETURN; // external stop was triggered
END_IF

IF OnHalt() THEN
  ; // Halting := TRUE; // Uncomment to acknowledge that the sequence is halting
END_IF

REPEAT
  LogStep();

  CASE _step.Index OF
    (* -------------------------------------------------------------------------------------------------------------------------------- *)
    MachineStep.GoHomeBegin:
    (* -------------------------------------------------------------------------------------------------------------------------------- *)
      IF _step.OnEntry()
      THEN
        _axis.ToolX.HomingAsync(THIS^);
        _axis.TransportX.HomingAsync(THIS^);  
			END_IF
      
      Await2(_axis.ToolX, _axis.TransportX, nextStep:=MachineStep.GoHomeEnd);

    (* -------------------------------------------------------------------------------------------------------------------------------- *)
    MachineStep.GoHomeEnd:
    (* -------------------------------------------------------------------------------------------------------------------------------- *)
      SetBusy(FALSE);
  
  ELSE
    Abort('sequence contains unhandled step');
  END_CASE
UNTIL _step.IsNotRepeatable() OR_ELSE NOT Busy END_REPEAT

END_FUNCTION_BLOCK

// ---- ZApp/Unit/Machine/_States/MachineSequenceFaultReaction.TcPOU
FUNCTION_BLOCK MachineSequenceFaultReaction EXTENDS MachineSequence IMPLEMENTS ZCore.ISequence
VAR
  _step : ZCore.Step(MachineStep.FaultReactionBegin, MachineStep.FaultReactionEnd);
  _timerSim : ZAux.Timer;
END_VAR

IF OnStart(_step) THEN
  ; // init custom sequence variables here ...
END_IF

REPEAT
  LogStep();

  CASE _step.Index OF
    (* -------------------------------------------------------------------------------------------------------------------------------- *)
    MachineStep.FaultReactionBegin:
    (* -------------------------------------------------------------------------------------------------------------------------------- *)
      IF _step.OnEntry()
      THEN
        _axis.TransportX.StopAsync(THIS^);
        _axis.ToolX.StopAsync(THIS^);        
			END_IF
      
      Await(_timerSim, nextStep:=MachineStep.FaultReactionEnd);
      // _step.SetNext(index:=MachineStep.FaultReactionEnd);

    (* -------------------------------------------------------------------------------------------------------------------------------- *)
    MachineStep.FaultReactionEnd:
    (* -------------------------------------------------------------------------------------------------------------------------------- *)    
      SetBusy(FALSE);
  
  ELSE
    Abort('sequence contains unhandled step');
  END_CASE
UNTIL _step.IsNotRepeatable() OR_ELSE NOT Busy END_REPEAT

END_FUNCTION_BLOCK

// ---- ZApp/Unit/Machine/MachineUnitProgram.TcPOU
/// each unit can run in its own PROGRAM and Task, respectively. However, this is optional and one may also
/// instantiate the unit in the ModuleProgram.
/// In order to keep initialization to a minimum, all ModuleContext objects that are required by the Unit are
/// given as FB_init parameter. These objects are
/// * data structs
/// * communication structs
/// * busmaster(s)
/// A unit should always be a root object (no parent) if it is running in its own context. If it runs in the same
/// task as the Module the parent may be set to the Module's Application.
PROGRAM MachineUnitProgram
VAR
{region "Machine"}
{undefine RunInSeparateProgram}
{IF NOT (defined (Machine_disabled)) AND (defined (RunInSeparateProgram))}
  Machine : MachineUnit(name := 'Machine', // name of the unit (for logging)
					  parent := 0, // caller of the Unit's cyclic method. If the Unit runs in its own context use 0
						configdata := ZGlobal.Data.Config.Machine,
						machinedata := ZGlobal.Data.Machine.Machine,
						calibrationdata := ZGlobal.Data.Calibration.Machine,
						com := ZGlobal.Com.Unit.Machine);
  {attribute 'section' := '__ZwPlcUnitProgramDeclaration__'}
  {attribute 'ZId' := 'ffcc16ae-32b8-4aad-8514-f391c00062a3'}
{END_IF}
{endregion}
{attribute '__ZwPlcUnitProgramDeclaration__'} // Do not remove this attribute! It is used for code generation.
END_VAR

// run the unit - the cylics of all children will be called as well

{region "Machine"}
{undefine RunInSeparateProgram}
{IF NOT (defined (Machine_disabled)) AND (defined (RunInSeparateProgram))}
  Machine.Cyclic();
  {attribute 'section' := '__ZwPlcUnitProgramImplementation__'}
  {attribute 'ZId' := 'ffcc16ae-32b8-4aad-8514-f391c00062a3'}
{END_IF}
{endregion}
{attribute '__ZwPlcUnitProgramImplementation__'} // Do not remove this attribute! It is used for code generation.

END_PROGRAM
